PROGRAM MAIN
VAR
	HEllo
END_VAR

END_PROGRAM

(* stored: Version 1.1.0.1, ProductVersion 3.1.4024.12
   POU MAIN: Id {41e3babf-3063-4e36-a1ee-fbfc92e8cfd0}, SpecialFunc None *)
